FUNCTION_BLOCK MIN_LWORD (* IEC 61131-3 LWORD Minimum *)
  (* Standard: 61131-3 *)
  (* Version 0.0, 2004-12-15, JHC, Rockwell Automation, Converted from SRC format. *)
  (* Compiler header: package fb.rt.plc.select; *)
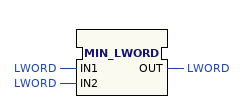
  VAR_INPUT
    IN1 : LWORD;
    IN2 : LWORD;
  END_VAR
  VAR_OUTPUT
    OUT : LWORD; (* MIN(IN1,IN2) *)
  END_VAR
END_FUNCTION_BLOCK
